# B&R Automation Studio project PO_MiRTS_Lab3
Automation Studio 4.5.2.102

## Configuration SampleText

### Task classes (Cpu.sw)
```
Cyclic#1 (cycle 2000 us, tolerance 0 us):
  SDCAxisCtr <- SDCAxisCtrlX.prg
DataObjects: Acp10sys
NcDataObjects: acp10etxen <- acp10etxen.dob, Axis_Xa <- Axis_Xobj.Axis_Xa.dob, Axis_Xi <- Axis_Xobj.Axis_Xi.dob
Binaries: udbdef, TCData, ashwd, ashwac, User, sysconf, asfw, arconfig, iomap, Role, Acp10map, acp10cfg
Libraries: Acp10sdc, sys_lib, Runtime, asstring, Acp10man, Acp10par, NcGlobal, Acp10_MC, brsystem, AsBrStr, Acp10sim, asieccon, powerlnk, astime, fileio, AsIOTime, MotorCtrl
```

### Hardware
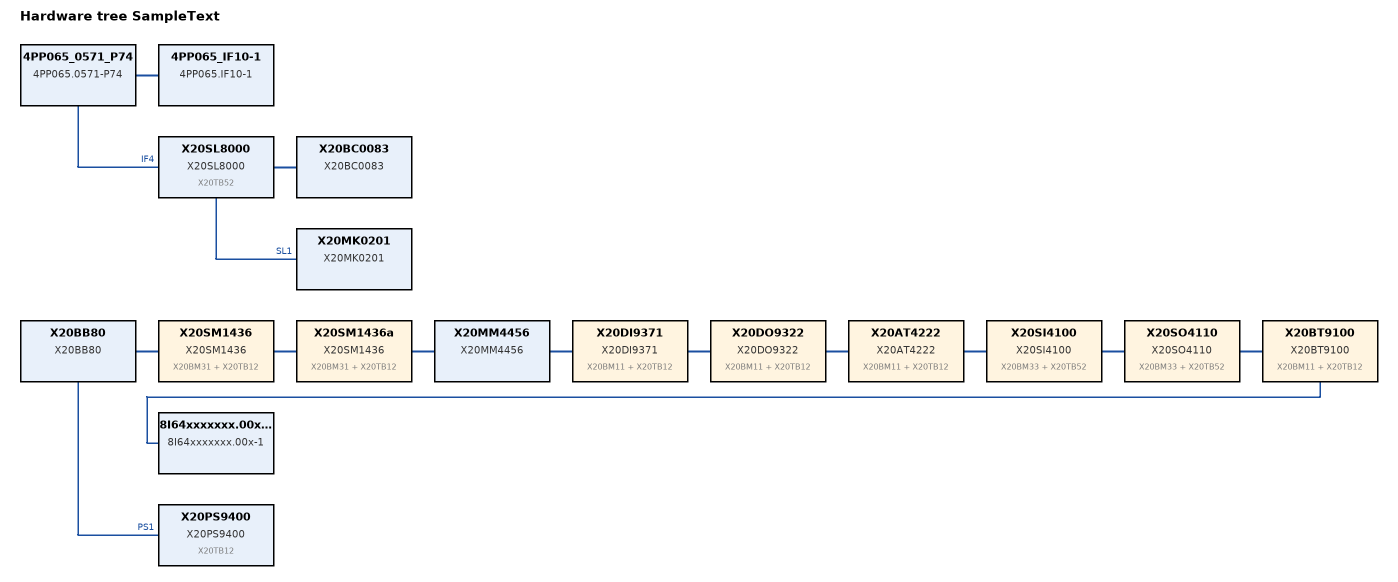
```
4PP065_0571_P74 : 4PP065.0571-P74 v1.1.2.0
  Connector IF4:
    EplInterfaceRedundant = 0
    EplEthInterfaceRedundant = 0
  Connector IF5:
    ActivateDevice = 1
    Mode = Manual
    InternetAddress = 10.1.1.13
    SubnetMask = 255.255.255.0
  ConfigurationID = DriveControl_SampleText
  TimerDeviceType = EPLX2X
  TimerDevice = 4PP065_0571_P74.IF4
  TaskClassIdleTime = 2000
  Cyclic1Duration = 2000
  Cyclic1Tolerance = 0
  Cyclic1Output = 1
4PP065_IF10-1 : 4PP065.IF10-1 v1.0.3.0  [SS -> 4PP065_0571_P74.SS1]
8I64xxxxxxx.00x-1 : 8I64xxxxxxx.00x-1 v1.3.9.1  [X2X1 -> X20BT9100.X2X1 [Cable Type=X2XCable, Length=10, Version=1.0.0.2]]
  ACC = 30
  DEC = 30
  UNS = 220
  NCR = 10
  NSP = 890
  COS = 64
  RSC = 33000
X20AT4222 : X20AT4222 v1.2.3.0  [SS1 -> X20TB12e.SS; SL -> X20BM11c.SL1]
X20BB80 : X20BB80 v1.0.2.0
X20BC0083 : X20BC0083 v2.9.0.0  [PLK1 -> X20SL8000.PLK2 (NodeNumber=2) [Cable Type=PowerlinkCable, Length=10, Version=1.0.0.2]; SL -> X20BB80.SL1]
X20BM11 : X20BM11 v1.0.0.1  [X2X1 -> X20BM33a.X2X2]
X20BM11a : X20BM11 v1.0.0.1  [X2X1 -> X20MM4456.X2X2]
X20BM11b : X20BM11 v1.0.0.1  [X2X1 -> X20BM11a.X2X2]
X20BM11c : X20BM11 v1.0.0.1  [X2X1 -> X20BM11b.X2X2]
X20BM31 : X20BM31 v1.0.0.1  [X2X1 -> X20BB80.IF1]
X20BM31a : X20BM31 v1.0.0.1  [X2X1 -> X20BM31.X2X2]
X20BM33 : X20BM33 v1.0.0.4  [X2X1 -> X20BM11c.X2X2]
X20BM33a : X20BM33 v1.0.0.4  [X2X1 -> X20BM33.X2X2]
X20BT9100 : X20BT9100 v1.0.3.0  [SS1 -> X20TB12f.SS; SL -> X20BM11.SL1]
X20DI9371 : X20DI9371 v1.0.2.0  [SS1 -> X20TB12c.SS; SL -> X20BM11a.SL1]
X20DO9322 : X20DO9322 v1.0.3.0  [SS1 -> X20TB12d.SS; SL -> X20BM11b.SL1]
X20MK0201 : X20MK0201 v1.0.0.0  [SL -> X20SL8000.SL1]
X20MM4456 : X20MM4456 v1.1.5.0  [X2X1 -> X20BM31a.X2X2]
X20PS9400 : X20PS9400 v1.0.2.4  [SS1 -> X20TB12.SS; PS -> X20BB80.PS1]
X20SI4100 : X20SI4100 v1.10.1.1  [SS1 -> X20TB52.SS; SL -> X20BM33.SL1]
X20SL8000 : X20SL8000 v1.6.5.1  [PLK1 -> 4PP065_0571_P74.IF4 (NodeNumber=1) [Cable Type=PowerlinkCable, Length=10, Version=1.0.0.2]; PLK2 -> X20BC0083.PLK1 (NodeNumber=1) [Cable Type=PowerlinkCable, Length=10, Version=1.0.0.2]; SS1 -> X20TB52b.SS]
  SafeProject = SafeLOGIC-1
X20SM1436 : X20SM1436 v1.4.2.1  [SS1 -> X20TB12a.SS; SL -> X20BM31.SL1]
X20SM1436a : X20SM1436 v1.4.2.1  [SS1 -> X20TB12b.SS; SL -> X20BM31a.SL1]
X20SO4110 : X20SO4110 v1.10.1.1  [SS1 -> X20TB52a.SS; SL -> X20BM33a.SL1]
  SafeModuleID = 3
X20TB12 : X20TB12 v1.0.0.0
X20TB12a : X20TB12 v1.0.0.0
X20TB12b : X20TB12 v1.0.0.0
X20TB12c : X20TB12 v1.0.0.0
X20TB12d : X20TB12 v1.0.0.0
X20TB12e : X20TB12 v1.0.0.0
X20TB12f : X20TB12 v1.0.0.0
X20TB52 : X20TB52 v1.0.0.1
X20TB52a : X20TB52 v1.0.0.1
X20TB52b : X20TB52 v1.0.0.1
```

### Acp10cfg.ncc - 4PP065_0571_P74/Motion/Acp10cfg.ncc
```
NcConfiguration (Version=5.02.1, NcSwId=Acp10)
  ACP10CF1_typ:
    cnt_nettrc_rec_drive = 1500
    bufsize_trace_upload = 1200
    tc_nc_man_task = Cyclic #1
    glob_pv_as_ncobject = Yes
    ncsys_dl_broadcast = Yes
    ncsys_dl_acp_reset = Yes
    safemc_log_err_to_ax = Yes
    network_init:
      ncsw_init_execute = Yes
      automatic_execute = No
      node_nr_warning = Yes
      net_err_before_ncact = Yes
    nettrc:
      enter_parsecrec = Yes
      enter_ncaction = Yes
      save_ring_startidx = Yes
    cam_prof_download:
      cam_dat_dl_parallel = No
      tc_cam_dl_parallel = Task class for NC Manager task
    plk_if[0]:
      if_name = IF4
      tc_CycDat_PLCopen = Task class for NC Manager task
      mc_broadcast_extdat = No
    sdc_if[0]:
      if_name = SDC_IF1
      mc_broadcast_size = 800
      mc_broadcast_extdat = No
```

### Acp10map.ncm - 4PP065_0571_P74/Motion/Acp10map.ncm
```
NcMapping (NcSwId=Acp10)
  NcObject Axis_X (ModuleId=8I64xxxxxxx.00x-1, ModuleAddress=SDC_IF1.ST1, Type=ncAXIS, Channel=1, AcoposSimulation=Off, InitParameter=Axis_Xi, AcoposParameter=Axis_Xa, Disabled=FALSE, ModuleDisabled=FALSE)
```

## Configuration Simulation

CPU , AutomationRuntime D4.52

## Logical view

Binary libraries used (declarations not repeated): Runtime, Operator, AsIecCon, astime, sys_lib, asstring, Acp10man, Acp10par, NcGlobal, Acp10sdc, Acp10_MC, brsystem, AsBrStr, Acp10sim, AsIOTime

### Global.var - Global variables
```iecst
VAR
	Axis_X : ACP10AXIS_typ := (0);
	Axis_X_HW : SdcHwCfg_typ := (0);
	Axis_X_DrvIf : SdcDrvIf16_typ := (0);
	Axis_X_DiDoIf : SdcDiDoIf_typ := (0);
	Axis_X_ModuleOk : BOOL := 0;
	Axis_X_EncIf : SdcEncIf16_typ := (0);
END_VAR
```

### Package Logical/Libraries - Global libraries

### Library Logical/Libraries/MotorCtrl (ANSIC)

#### Constants.var - Exported constants
```iecst
VAR CONSTANT
	COUNTER_BUFFER_CYCLES : USINT := 64;
	UNITS_PER_ROTATION : REAL := 3000;
END_VAR
```

#### MotorCtrl.fun - Exported functions and function blocks
```iecst
{REDUND_ERROR} {REDUND_UNREPLICABLE} FUNCTION_BLOCK FB_Integrator (*TODO: Add your comment here*) (*$GROUP=User,$CAT=User,$GROUPICON=User.png,$CATICON=User.png*)
	VAR_INPUT
		in : {REDUND_UNREPLICABLE} REAL;
	END_VAR
	VAR_OUTPUT
		out : {REDUND_UNREPLICABLE} REAL;
	END_VAR
	VAR
		dt : {REDUND_UNREPLICABLE} REAL;
		state : {REDUND_UNREPLICABLE} REAL;
	END_VAR
END_FUNCTION_BLOCK

{REDUND_ERROR} FUNCTION_BLOCK FB_Motor (*TODO: Add your comment here*) (*$GROUP=User,$CAT=User,$GROUPICON=User.png,$CATICON=User.png*)
	VAR_INPUT
		u : {REDUND_UNREPLICABLE} REAL;
	END_VAR
	VAR_OUTPUT
		phi : {REDUND_UNREPLICABLE} REAL;
		w : REAL;
	END_VAR
	VAR
		integrator2 : {REDUND_UNREPLICABLE} FB_Integrator;
		Tm : {REDUND_UNREPLICABLE} REAL;
		ke : {REDUND_UNREPLICABLE} REAL;
		dt : {REDUND_UNREPLICABLE} REAL;
		integrator1 : FB_Integrator;
	END_VAR
END_FUNCTION_BLOCK

{REDUND_ERROR} {REDUND_UNREPLICABLE} FUNCTION_BLOCK FB_Regulator (*TODO: Add your comment here*) (*$GROUP=User,$CAT=User,$GROUPICON=User.png,$CATICON=User.png*)
	VAR_INPUT
		e : {REDUND_UNREPLICABLE} REAL;
	END_VAR
	VAR_OUTPUT
		u : {REDUND_UNREPLICABLE} REAL;
	END_VAR
	VAR
		k_p : {REDUND_UNREPLICABLE} REAL;
		k_i : {REDUND_UNREPLICABLE} REAL;
		integrator : {REDUND_UNREPLICABLE} FB_Integrator;
		iyOld : {REDUND_UNREPLICABLE} REAL;
		max_abs_value : {REDUND_UNREPLICABLE} REAL;
		dt : {REDUND_UNREPLICABLE} REAL;
	END_VAR
END_FUNCTION_BLOCK

{REDUND_ERROR} FUNCTION_BLOCK FB_Axis (* *) (*$GROUP=User,$CAT=User,$GROUPICON=User.png,$CATICON=User.png*)
	VAR_INPUT
		reset_error : {REDUND_UNREPLICABLE} BOOL;
		endswitch_a_reached : {REDUND_UNREPLICABLE} BOOL;
		endswitch_b_reached : {REDUND_UNREPLICABLE} BOOL;
		pwm_period : REAL;
		counter : DINT;
	END_VAR
	VAR_OUTPUT
		reset_counter : {REDUND_UNREPLICABLE} BOOL;
		pwm_value : {REDUND_UNREPLICABLE} REAL;
		speed : {REDUND_UNREPLICABLE} REAL;
	END_VAR
	VAR
		last_counter : {REDUND_UNREPLICABLE} DINT;
		regulator : FB_Regulator;
		desired_speed : REAL;
		counter_buffer : INT := 0;
	END_VAR
END_FUNCTION_BLOCK
```

#### FB_Motor.c
```c
#include <bur/plctypes.h>
#ifdef __cplusplus
	extern "C"
	{
#endif
	#include "MotorCtrl.h"
#ifdef __cplusplus
	};
#endif
/* TODO: Add your comment here */
void FB_Motor(struct FB_Motor* inst)
{
	/*TODO: Add your code here*/
	REAL a = inst->u / inst->ke - inst->w;

	inst->integrator1.in = a;
	FB_Integrator(&inst->integrator1);
	inst->w = inst->integrator1.out;

	inst->integrator2.in = inst->w;
	FB_Integrator(&inst->integrator2);
	inst->phi = inst->integrator2.out;
}
```

#### FB_Integrator.c
```c
#include <bur/plctypes.h>
#ifdef __cplusplus
	extern "C"
	{
#endif
	#include "MotorCtrl.h"
#ifdef __cplusplus
	};
#endif
/* TODO: Add your comment here */
void FB_Integrator(struct FB_Integrator* inst)
{
	inst->out = inst->dt * inst->in + inst->state;
	inst->state = inst->out;
}
```

#### FB_Regulator.c
```c
#include <bur/plctypes.h>
#ifdef __cplusplus
	extern "C"
	{
#endif
	#include "MotorCtrl.h"
#ifdef __cplusplus
	};
#endif

void FB_Regulator(struct FB_Regulator* inst)
{
	REAL a = inst->e * inst->k_p;
	REAL b = inst->e * inst->k_i;
	a = a > inst->max_abs_value ? inst->max_abs_value : a;
	a = a < -inst->max_abs_value ? -inst->max_abs_value : a;
	inst->integrator.in = b + inst->iyOld;
	FB_Integrator(&inst->integrator);
	REAL sum = a + inst->integrator.out;
	inst->u = sum;
	inst->u = inst->u > inst->max_abs_value ? inst->max_abs_value : inst->u;
	inst->u = inst->u < -inst->max_abs_value ? -inst->max_abs_value : inst->u;
	inst->iyOld = inst->u - sum;
}
```

#### FB_Axis.c
```c
#include <bur/plctypes.h>
#ifdef __cplusplus
	extern "C"
	{
#endif
	#include "MotorCtrl.h"
#ifdef __cplusplus
	};
#endif
#ifdef _DEFAULT_INCLUDES
	#include <AsDefault.h>
#endif

void FB_Axis(struct FB_Axis* inst)
{
	inst->counter_buffer += inst->counter - inst->last_counter;
	inst->last_counter = inst->counter;
	Axis_X_EncIf.iActPos = inst->counter;
	if((Axis_X_EncIf.iLifeCnt) % COUNTER_BUFFER_CYCLES == 0){
		inst->speed = (inst->counter_buffer) / (0.002 * COUNTER_BUFFER_CYCLES); // cycle = 2 ms
		inst->counter_buffer = 0;
	}
	Axis_X_DiDoIf.iNegHwEnd = inst->endswitch_a_reached;
	Axis_X_DiDoIf.iPosHwEnd = inst->endswitch_b_reached;
	inst->desired_speed = Axis_X_DrvIf.oSetPos * UNITS_PER_ROTATION / 32767;
	inst->regulator.e = inst->desired_speed - inst->speed;
	FB_Regulator(&(inst->regulator));
	inst->pwm_value = (inst->regulator.u) / (inst->regulator.max_abs_value) * (inst->pwm_period);
}
```

### Package Logical/Axis_Xobj - Axis_Xobj

### Data object Logical/Axis_Xobj/Axis_Xa (Apt)

#### Axis_Xa.apt
```
AcoposParameterTable:
  Root Parameters:
    230 = PCTRL_S_SET (Name=PCTRL_S_ACT_PARID)
    109 = 24 (Name=SCALE_ENCOD_INCR)  // Encoder1: Encoder scaling: increments per encoder revolution
    64201 = 6500 (Name=SERVO_V_MAX_OUTPUT)
```

### Data object Logical/Axis_Xobj/Axis_Xi (Ax)

#### Axis_Xi.ax
```
InitParameter (Version=5.2.1, NcSwId=ACP10)
  ACP10AXIS_typ:
    dig_in:
      level:
        reference = ncACTIV_HI
        pos_hw_end = ncACTIV_HI
        neg_hw_end = ncACTIV_HI
        trigger1 = ncACTIV_HI
        trigger2 = ncACTIV_HI
    encoder_if:
      parameter:
        count_dir = ncSTANDARD
        scaling:
          load:
            units = 3000
            rev_motor = 1
    limit:
      parameter:
        v_pos = 10000.0
        v_neg = 10000.0
        a1_pos = 10000.0
        a2_pos = 10000.0
        a1_neg = 10000.0
        a2_neg = 10000.0
        t_jolt = 0.0
        t_in_pos = 0.0
        pos_sw_end = 8388607
        neg_sw_end = -8388608
        ds_warning = 500.0
        ds_stop = 50000.0
        a_stop = 1.0E+30
        dv_stop = 0.0
        dv_stop_mode = ncOFF
    controller:
      mode = ncPOSITION
      position:
        kv = 10.0
        tn = 0.0
        t_predict = 0.01
        t_total = 0.01
        p_max = 1.0E+30
        i_max = 0.0
      speed:
        kv = 2.0
        tn = 0.0
        t_filter = 0.0
        isq_filter1:
          type = ncOFF
          a0 = 0.0
          a1 = 0.0
          b0 = 0.0
          b1 = 0.0
          b2 = 0.0
          c0_par_id = 0
          c1_par_id = 0
        isq_filter2:
          type = ncOFF
          a0 = 0.0
          a1 = 0.0
          b0 = 0.0
          b1 = 0.0
          b2 = 0.0
          c0_par_id = 0
          c1_par_id = 0
        isq_filter3:
          type = ncOFF
          a0 = 0.0
          a1 = 0.0
          b0 = 0.0
          b1 = 0.0
          b2 = 0.0
          c0_par_id = 0
          c1_par_id = 0
      uf:
        type = ncLINEAR + ncCORRECTION
        auto_config = ncMOTOR_PAR
        u0 = 0.0
        un = 0.0
        fn = 50.0
        k_f_slip = 0.0
      ff:
        torque_load = 0.0
        torque_pos = 0.0
        torque_neg = 0.0
        kv_torque = 0.0
        inertia = 0.0
        t_filter_a = 0.0
    move:
      stop:
        parameter[0]:
          decel_ramp = ncA_LIMIT
          controller = ncON
        parameter[1]:
          decel_ramp = ncA_LIMIT
          controller = ncON
        parameter[2]:
          decel_ramp = ncA_LIMIT
          controller = ncON
        parameter[3]:
          decel_ramp = ncA_LIMIT
          controller = ncON
        quickstop:
          decel_ramp = ncA_LIMIT
          t_jolt = 0.0
        drive_error:
          decel_ramp = ncA_LIMIT
      homing:
        parameter:
          s = 0
          v_switch = 6000.0
          v_trigger = 2000.0
          a = 10000.0
          mode = ncEND_SWITCH
          edge_sw = ncNEGATIVE
          start_dir = ncPOSITIVE
          trigg_dir = ncNEGATIVE
          ref_pulse = ncOFF
          fix_dir = ncOFF
          tr_s_block = 0.0
          torque_lim = 0.0
          ds_block = 0.0
          ds_stop = 0.0
      basis:
        parameter:
          v_pos = 6000.0
          v_neg = 6000.0
          a1_pos = 10000.0
          a2_pos = 10000.0
          a1_neg = 10000.0
          a2_neg = 10000.0
    message:
      text:
        parameter:
          format = ncBREAK
          columns = 80
          data_modul = acp10etxen
```

### Program Logical/SDCAxisCtrlX (ANSIC)

#### Variables.var
```iecst
VAR
	motor_X : FB_Motor := (0);
	pwm_period : REAL := 0.0;
	coil_pwm_value : INT := 0;
	coil_powered : BOOL := FALSE;
	axis_X : FB_Axis := (0);
END_VAR
VAR CONSTANT
	MAX_UNITS_PER_SECOND : UINT := 6500;
END_VAR
```

#### Main.c
```c
#include <bur/plctypes.h>

#ifdef _DEFAULT_INCLUDES
	#include <AsDefault.h>
#endif

void _INIT ProgramInit(void)
{
	Axis_X_HW.EncIf1_Typ = ncSDC_ENC16;
	Axis_X_HW.DiDoIf_Typ = ncSDC_DIDO;
	Axis_X_HW.DrvIf_Typ = ncSDC_DRVSERVO16;
	strcpy(Axis_X_HW.EncIf1_Name, "Axis_X_EncIf");
	strcpy(Axis_X_HW.DrvIf_Name, "Axis_X_DrvIf");
	strcpy(Axis_X_HW.DiDoIf_Name, "Axis_X_DiDoIf");

	Axis_X_ModuleOk = 1;
	Axis_X_EncIf.iEncOK = 1;
	Axis_X_DrvIf.iDrvOK = 1;
	Axis_X_DrvIf.iStatusEnable = 1;
	Axis_X_DiDoIf.iDriveReady = 1;

	axis_X.counter = axis_X.last_counter = 0;
	axis_X.pwm_period = pwm_period = 0.05;
	axis_X.regulator.dt = 0.002;
	axis_X.regulator.integrator.dt = 0.002;
	axis_X.regulator.k_i = 0.0072;
	axis_X.regulator.k_p = 0.0072;
	axis_X.regulator.max_abs_value = 24.0;

	motor_X.dt = 0.01;
	motor_X.ke = 1;
	motor_X.Tm = 0.1;
	motor_X.u = 0;
	motor_X.phi = 0;
	motor_X.integrator1.dt = 0.002 / motor_X.Tm;
	motor_X.integrator2.dt = 0.002;
}

void _CYCLIC ProgramCyclic(void)
{
	Axis_X_EncIf.iLifeCnt++;
	Axis_X_EncIf.iActTime = (INT)AsIOTimeCyclicStart();
	Axis_X_DrvIf.iLifeCnt++;
	Axis_X_DrvIf.oSetPos = Axis_X.monitor.v;
	Axis_X_DiDoIf.iLifeCntDriveEnable++;
	Axis_X_DiDoIf.iLifeCntDriveReady++;
	Axis_X_DiDoIf.iLifeCntNegHwEnd++;
	Axis_X_DiDoIf.iLifeCntPosHwEnd++;
	Axis_X_DiDoIf.iLifeCntReference++;
	FB_Axis(&axis_X);
	if(Axis_X_DrvIf.oSetPos != 0){
		motor_X.u = axis_X.pwm_value / axis_X.pwm_period * MAX_UNITS_PER_SECOND;
		FB_Motor(&motor_X);
		axis_X.counter = motor_X.phi;
		if (axis_X.counter <= -3000)
			axis_X.endswitch_a_reached = 1;
		else
			axis_X.endswitch_a_reached = 0;
		if (axis_X.counter >= 3000)
			axis_X.endswitch_b_reached = 1;
		else
			axis_X.endswitch_b_reached = 0;
	}
}

void _EXIT ProgramExit(void)
{

}
```

Listed in the project but not available here: Logical/Global.typ, Logical/Libraries/MotorCtrl/Variables.var, Logical/acp10etxen
